// TIA Portal V20 export
FUNCTION "FC_Sequenza_Start" : Void   // FC300, LAD
{ S7_Optimized_Access := 'TRUE' }
// stored: AutoNumber false, SetENOAutomatically false
   VAR_TEMP   // added for the SCL form of the ladder/FBD networks
      _w1 : Bool;
      _w2 : Bool;
      _w3 : Bool;
      _w4 : Bool;
      _w5 : Bool;
      _w6 : Bool;
      _w7 : Bool;
      _w8 : Bool;
      _w9 : Bool;
      _w10 : Bool;
   END_VAR
BEGIN

REGION Network 1: Controllo ventilatori zona 1
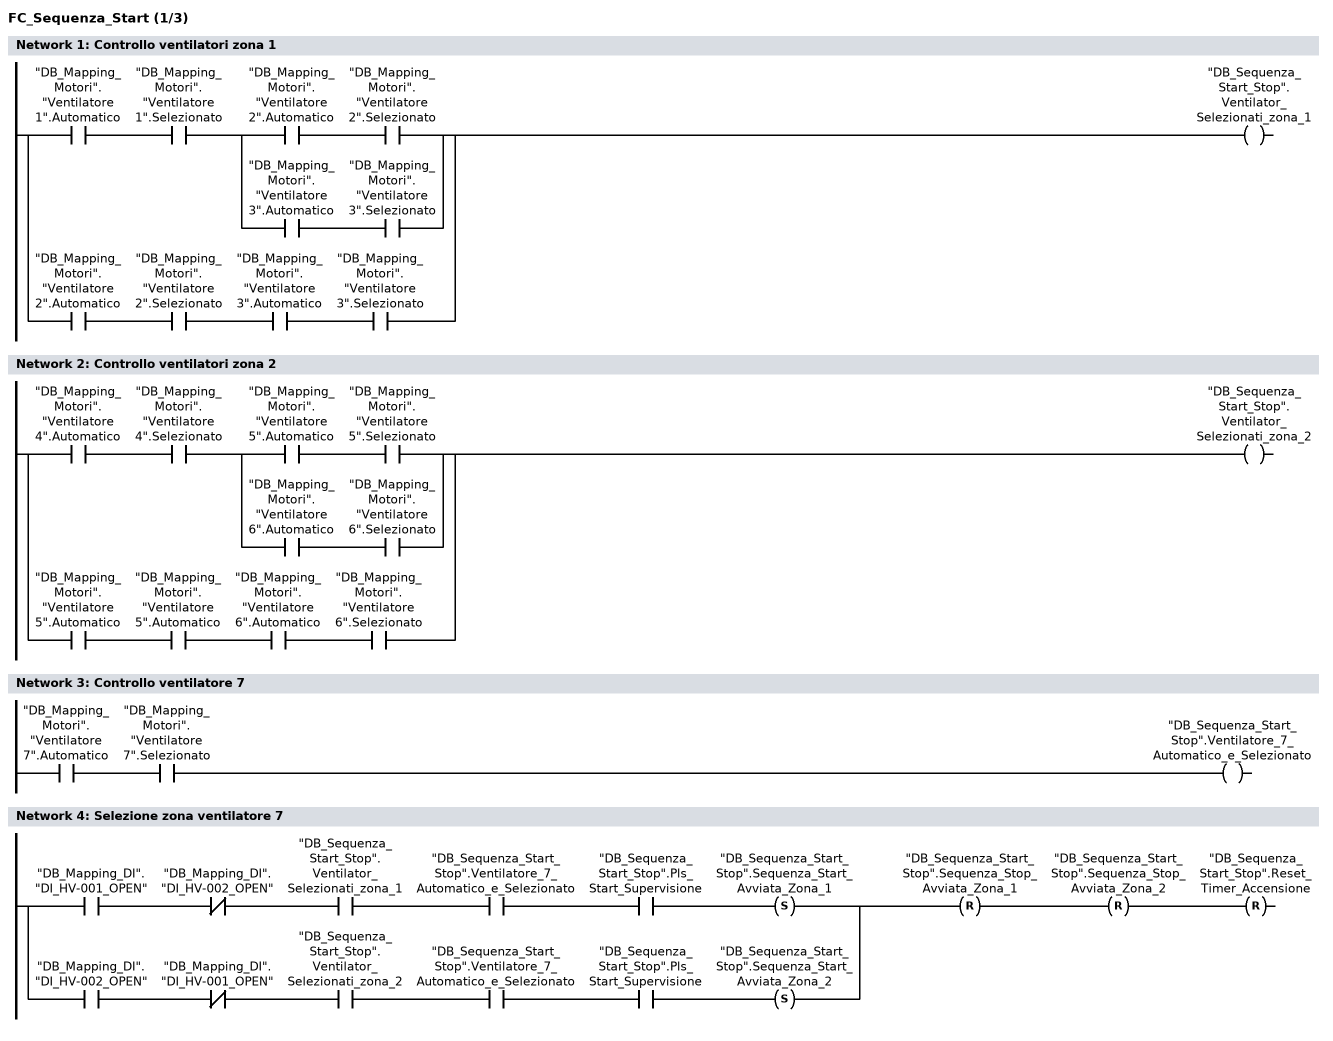
   RUNG wire#powerrail
      Contact( "DB_Mapping_Motori"."Ventilatore 1".Automatico )
      Contact( "DB_Mapping_Motori"."Ventilatore 1".Selezionato )
      wire#w1
      Contact( "DB_Mapping_Motori"."Ventilatore 2".Automatico )
      Contact( "DB_Mapping_Motori"."Ventilatore 2".Selezionato )
      wire#w2
      Coil( "DB_Sequenza_Start_Stop".Ventilator_Selezionati_zona_1 )
   END_RUNG
   RUNG wire#w1
      Contact( "DB_Mapping_Motori"."Ventilatore 3".Automatico )
      Contact( "DB_Mapping_Motori"."Ventilatore 3".Selezionato )
   END_RUNG wire#w2
   RUNG wire#powerrail
      Contact( "DB_Mapping_Motori"."Ventilatore 2".Automatico )
      Contact( "DB_Mapping_Motori"."Ventilatore 2".Selezionato )
      Contact( "DB_Mapping_Motori"."Ventilatore 3".Automatico )
      Contact( "DB_Mapping_Motori"."Ventilatore 3".Selezionato )
   END_RUNG wire#w2
   // the same network as SCL:
   "DB_Sequenza_Start_Stop".Ventilator_Selezionati_zona_1 := ("DB_Mapping_Motori"."Ventilatore 1".Automatico AND "DB_Mapping_Motori"."Ventilatore 1".Selezionato AND (("DB_Mapping_Motori"."Ventilatore 2".Automatico AND "DB_Mapping_Motori"."Ventilatore 2".Selezionato) OR ("DB_Mapping_Motori"."Ventilatore 3".Automatico AND "DB_Mapping_Motori"."Ventilatore 3".Selezionato))) OR ("DB_Mapping_Motori"."Ventilatore 2".Automatico AND "DB_Mapping_Motori"."Ventilatore 2".Selezionato AND "DB_Mapping_Motori"."Ventilatore 3".Automatico AND "DB_Mapping_Motori"."Ventilatore 3".Selezionato);
END_REGION

REGION Network 2: Controllo ventilatori zona 2
   RUNG wire#powerrail
      Contact( "DB_Mapping_Motori"."Ventilatore 4".Automatico )
      Contact( "DB_Mapping_Motori"."Ventilatore 4".Selezionato )
      wire#w1
      Contact( "DB_Mapping_Motori"."Ventilatore 5".Automatico )
      Contact( "DB_Mapping_Motori"."Ventilatore 5".Selezionato )
      wire#w2
      Coil( "DB_Sequenza_Start_Stop".Ventilator_Selezionati_zona_2 )
   END_RUNG
   RUNG wire#w1
      Contact( "DB_Mapping_Motori"."Ventilatore 6".Automatico )
      Contact( "DB_Mapping_Motori"."Ventilatore 6".Selezionato )
   END_RUNG wire#w2
   RUNG wire#powerrail
      Contact( "DB_Mapping_Motori"."Ventilatore 5".Automatico )
      Contact( "DB_Mapping_Motori"."Ventilatore 5".Automatico )
      Contact( "DB_Mapping_Motori"."Ventilatore 6".Automatico )
      Contact( "DB_Mapping_Motori"."Ventilatore 6".Selezionato )
   END_RUNG wire#w2
   // the same network as SCL:
   "DB_Sequenza_Start_Stop".Ventilator_Selezionati_zona_2 := ("DB_Mapping_Motori"."Ventilatore 4".Automatico AND "DB_Mapping_Motori"."Ventilatore 4".Selezionato AND (("DB_Mapping_Motori"."Ventilatore 5".Automatico AND "DB_Mapping_Motori"."Ventilatore 5".Selezionato) OR ("DB_Mapping_Motori"."Ventilatore 6".Automatico AND "DB_Mapping_Motori"."Ventilatore 6".Selezionato))) OR ("DB_Mapping_Motori"."Ventilatore 5".Automatico AND "DB_Mapping_Motori"."Ventilatore 5".Automatico AND "DB_Mapping_Motori"."Ventilatore 6".Automatico AND "DB_Mapping_Motori"."Ventilatore 6".Selezionato);
END_REGION

REGION Network 3: Controllo ventilatore 7
   RUNG wire#powerrail
      Contact( "DB_Mapping_Motori"."Ventilatore 7".Automatico )
      Contact( "DB_Mapping_Motori"."Ventilatore 7".Selezionato )
      Coil( "DB_Sequenza_Start_Stop".Ventilatore_7_Automatico_e_Selezionato )
   END_RUNG
   // the same network as SCL:
   "DB_Sequenza_Start_Stop".Ventilatore_7_Automatico_e_Selezionato := "DB_Mapping_Motori"."Ventilatore 7".Automatico AND "DB_Mapping_Motori"."Ventilatore 7".Selezionato;
END_REGION

REGION Network 4: Selezione zona ventilatore 7
   RUNG wire#powerrail
      Contact( "DB_Mapping_DI"."DI_HV-001_OPEN" )
      I_Contact( "DB_Mapping_DI"."DI_HV-002_OPEN" )
      Contact( "DB_Sequenza_Start_Stop".Ventilator_Selezionati_zona_1 )
      Contact( "DB_Sequenza_Start_Stop".Ventilatore_7_Automatico_e_Selezionato )
      Contact( "DB_Sequenza_Start_Stop".Pls_Start_Supervisione )
      S_Coil( "DB_Sequenza_Start_Stop".Sequenza_Start_Avviata_Zona_1 )
      wire#w1
      R_Coil( "DB_Sequenza_Start_Stop".Sequenza_Stop_Avviata_Zona_1 )
      R_Coil( "DB_Sequenza_Start_Stop".Sequenza_Stop_Avviata_Zona_2 )
      R_Coil( "DB_Sequenza_Start_Stop".Reset_Timer_Accensione )
   END_RUNG
   RUNG wire#powerrail
      Contact( "DB_Mapping_DI"."DI_HV-002_OPEN" )
      I_Contact( "DB_Mapping_DI"."DI_HV-001_OPEN" )
      Contact( "DB_Sequenza_Start_Stop".Ventilator_Selezionati_zona_2 )
      Contact( "DB_Sequenza_Start_Stop".Ventilatore_7_Automatico_e_Selezionato )
      Contact( "DB_Sequenza_Start_Stop".Pls_Start_Supervisione )
      S_Coil( "DB_Sequenza_Start_Stop".Sequenza_Start_Avviata_Zona_2 )
   END_RUNG wire#w1
   // the same network as SCL:
   #_w1 := "DB_Mapping_DI"."DI_HV-001_OPEN" AND NOT "DB_Mapping_DI"."DI_HV-002_OPEN" AND "DB_Sequenza_Start_Stop".Ventilator_Selezionati_zona_1 AND "DB_Sequenza_Start_Stop".Ventilatore_7_Automatico_e_Selezionato AND "DB_Sequenza_Start_Stop".Pls_Start_Supervisione;
   IF #_w1 THEN "DB_Sequenza_Start_Stop".Sequenza_Start_Avviata_Zona_1 := TRUE; END_IF;
   #_w2 := "DB_Mapping_DI"."DI_HV-002_OPEN" AND NOT "DB_Mapping_DI"."DI_HV-001_OPEN" AND "DB_Sequenza_Start_Stop".Ventilator_Selezionati_zona_2 AND "DB_Sequenza_Start_Stop".Ventilatore_7_Automatico_e_Selezionato AND "DB_Sequenza_Start_Stop".Pls_Start_Supervisione;
   IF #_w2 THEN "DB_Sequenza_Start_Stop".Sequenza_Start_Avviata_Zona_2 := TRUE; END_IF;
   IF #_w1 OR #_w2 THEN
       "DB_Sequenza_Start_Stop".Sequenza_Stop_Avviata_Zona_1 := FALSE;
       "DB_Sequenza_Start_Stop".Sequenza_Stop_Avviata_Zona_2 := FALSE;
       "DB_Sequenza_Start_Stop".Reset_Timer_Accensione := FALSE;
   END_IF;
END_REGION

REGION Network 5: Accensione ventilatori
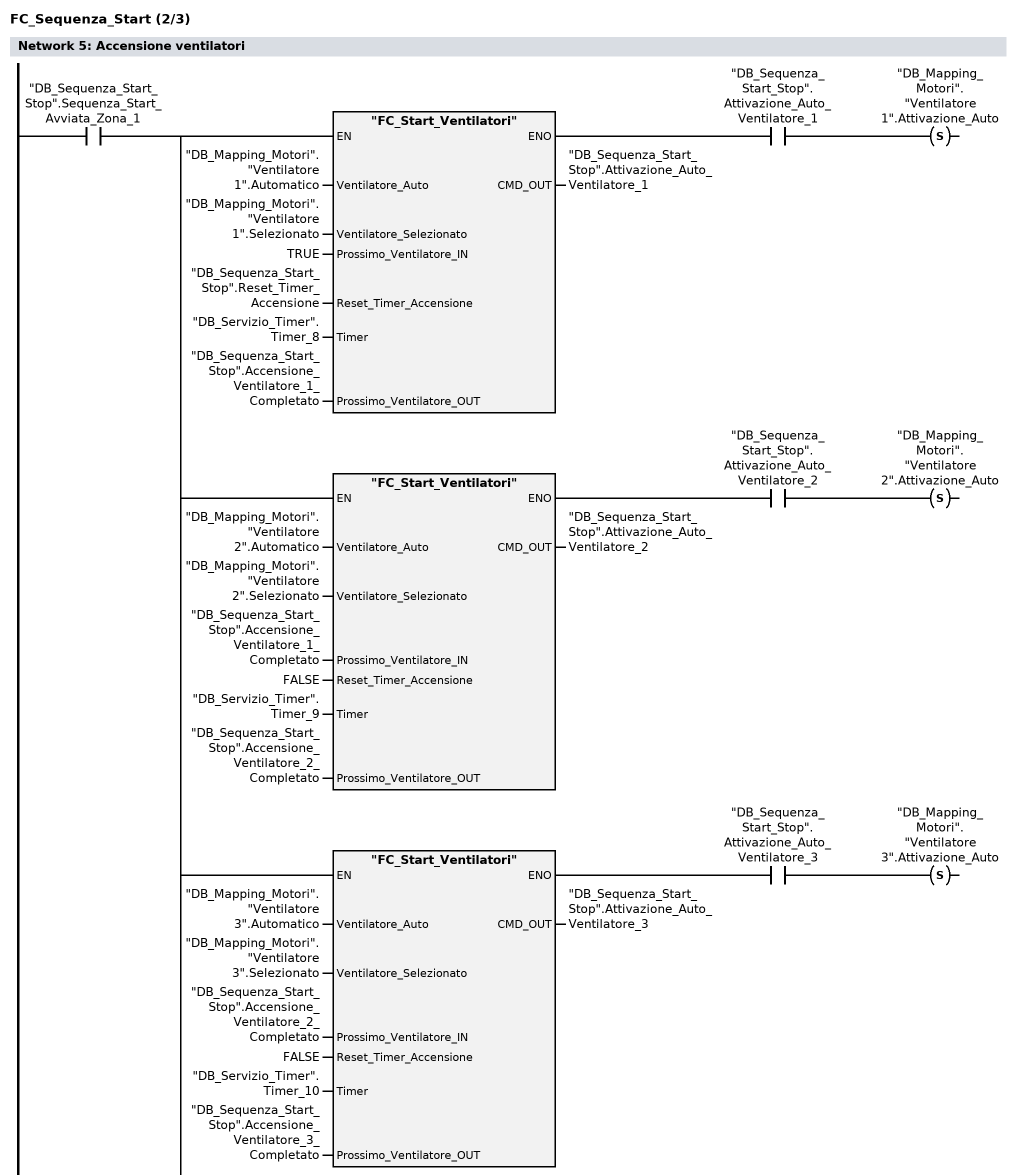
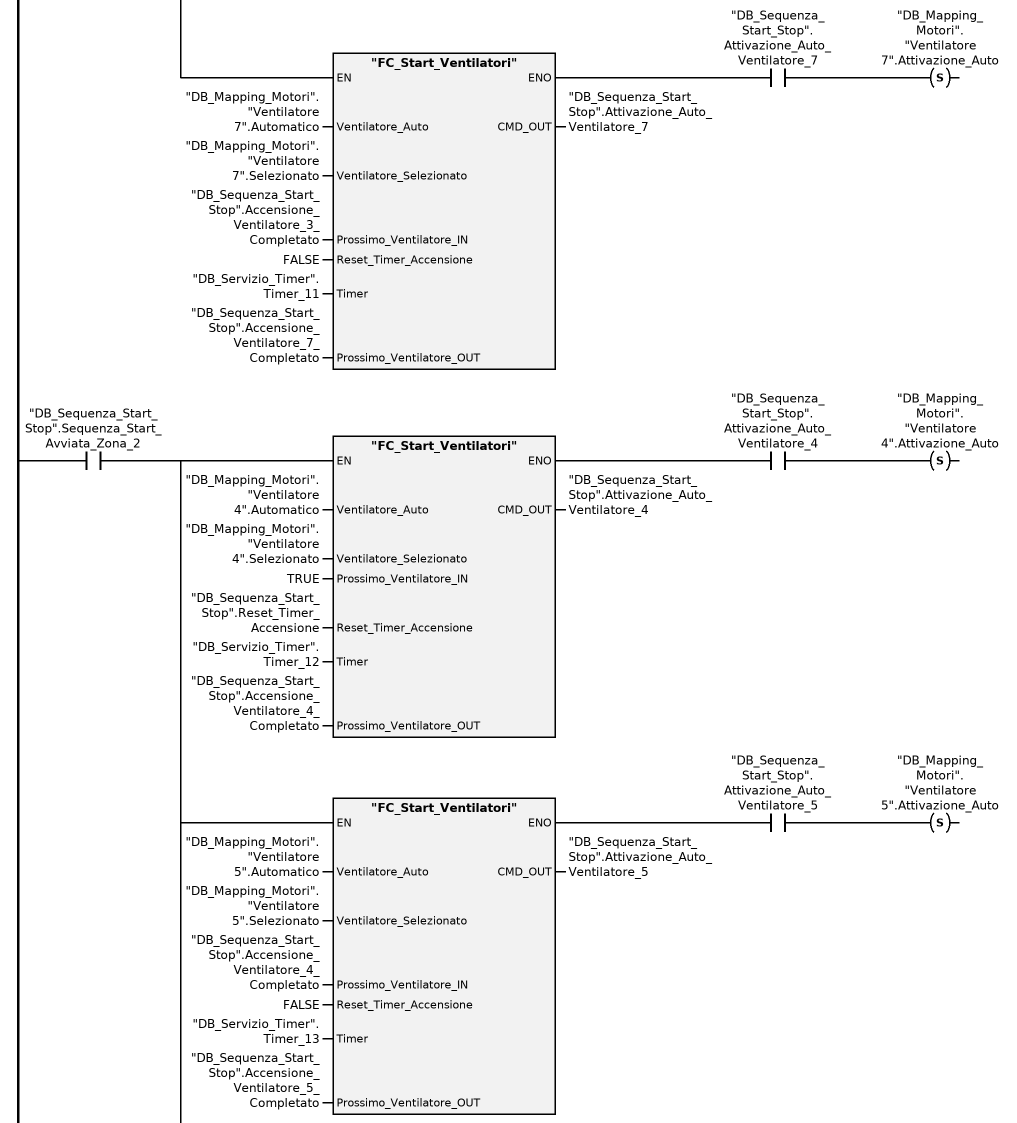
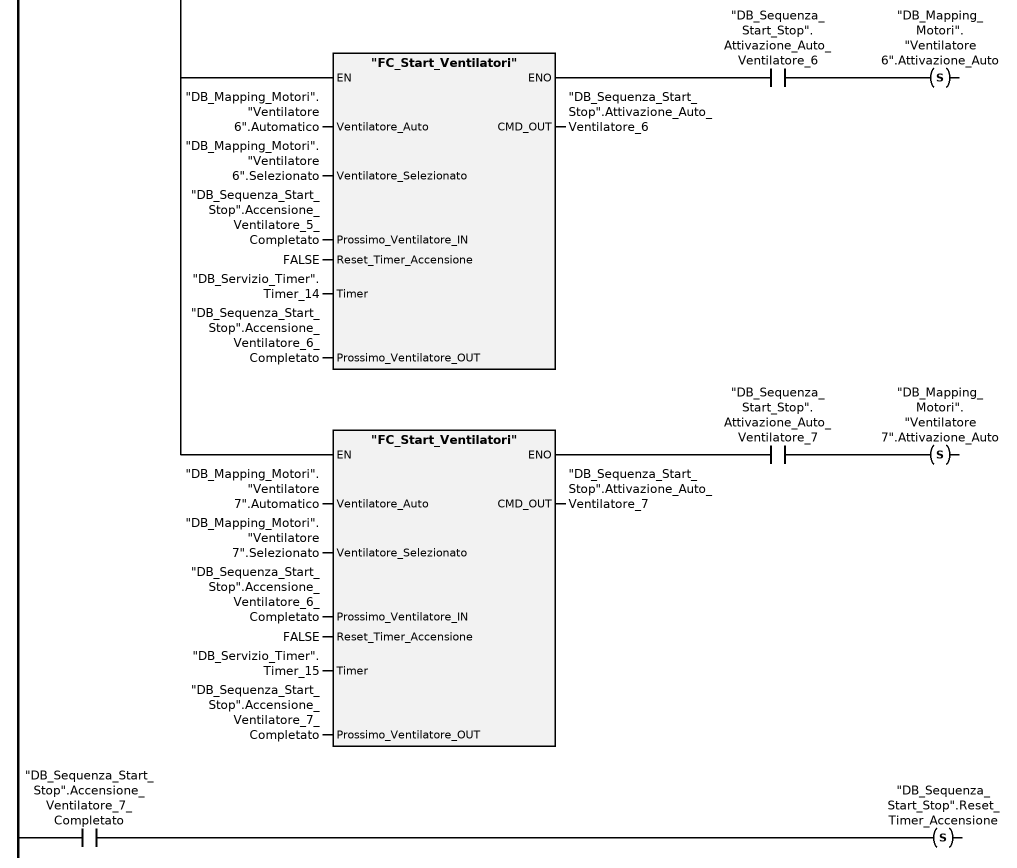
   RUNG wire#powerrail
      Contact( "DB_Sequenza_Start_Stop".Sequenza_Start_Avviata_Zona_1 )
      wire#w1
      "FC_Start_Ventilatori"(Ventilatore_Auto := "DB_Mapping_Motori"."Ventilatore 1".Automatico, Ventilatore_Selezionato := "DB_Mapping_Motori"."Ventilatore 1".Selezionato, Prossimo_Ventilatore_IN := TRUE, Reset_Timer_Accensione := "DB_Sequenza_Start_Stop".Reset_Timer_Accensione, "Timer" := "DB_Servizio_Timer".Timer_8, Prossimo_Ventilatore_OUT := "DB_Sequenza_Start_Stop".Accensione_Ventilatore_1_Completato, CMD_OUT => "DB_Sequenza_Start_Stop".Attivazione_Auto_Ventilatore_1)
      Contact( "DB_Sequenza_Start_Stop".Attivazione_Auto_Ventilatore_1 )
      S_Coil( "DB_Mapping_Motori"."Ventilatore 1".Attivazione_Auto )
   END_RUNG
   RUNG wire#w1
      "FC_Start_Ventilatori"(Ventilatore_Auto := "DB_Mapping_Motori"."Ventilatore 2".Automatico, Ventilatore_Selezionato := "DB_Mapping_Motori"."Ventilatore 2".Selezionato, Prossimo_Ventilatore_IN := "DB_Sequenza_Start_Stop".Accensione_Ventilatore_1_Completato, Reset_Timer_Accensione := FALSE, "Timer" := "DB_Servizio_Timer".Timer_9, Prossimo_Ventilatore_OUT := "DB_Sequenza_Start_Stop".Accensione_Ventilatore_2_Completato, CMD_OUT => "DB_Sequenza_Start_Stop".Attivazione_Auto_Ventilatore_2)
      Contact( "DB_Sequenza_Start_Stop".Attivazione_Auto_Ventilatore_2 )
      S_Coil( "DB_Mapping_Motori"."Ventilatore 2".Attivazione_Auto )
   END_RUNG
   RUNG wire#w1
      "FC_Start_Ventilatori"(Ventilatore_Auto := "DB_Mapping_Motori"."Ventilatore 3".Automatico, Ventilatore_Selezionato := "DB_Mapping_Motori"."Ventilatore 3".Selezionato, Prossimo_Ventilatore_IN := "DB_Sequenza_Start_Stop".Accensione_Ventilatore_2_Completato, Reset_Timer_Accensione := FALSE, "Timer" := "DB_Servizio_Timer".Timer_10, Prossimo_Ventilatore_OUT := "DB_Sequenza_Start_Stop".Accensione_Ventilatore_3_Completato, CMD_OUT => "DB_Sequenza_Start_Stop".Attivazione_Auto_Ventilatore_3)
      Contact( "DB_Sequenza_Start_Stop".Attivazione_Auto_Ventilatore_3 )
      S_Coil( "DB_Mapping_Motori"."Ventilatore 3".Attivazione_Auto )
   END_RUNG
   RUNG wire#w1
      "FC_Start_Ventilatori"(Ventilatore_Auto := "DB_Mapping_Motori"."Ventilatore 7".Automatico, Ventilatore_Selezionato := "DB_Mapping_Motori"."Ventilatore 7".Selezionato, Prossimo_Ventilatore_IN := "DB_Sequenza_Start_Stop".Accensione_Ventilatore_3_Completato, Reset_Timer_Accensione := FALSE, "Timer" := "DB_Servizio_Timer".Timer_11, Prossimo_Ventilatore_OUT := "DB_Sequenza_Start_Stop".Accensione_Ventilatore_7_Completato, CMD_OUT => "DB_Sequenza_Start_Stop".Attivazione_Auto_Ventilatore_7)
      Contact( "DB_Sequenza_Start_Stop".Attivazione_Auto_Ventilatore_7 )
      S_Coil( "DB_Mapping_Motori"."Ventilatore 7".Attivazione_Auto )
   END_RUNG
   RUNG wire#powerrail
      Contact( "DB_Sequenza_Start_Stop".Sequenza_Start_Avviata_Zona_2 )
      wire#w2
      "FC_Start_Ventilatori"(Ventilatore_Auto := "DB_Mapping_Motori"."Ventilatore 4".Automatico, Ventilatore_Selezionato := "DB_Mapping_Motori"."Ventilatore 4".Selezionato, Prossimo_Ventilatore_IN := TRUE, Reset_Timer_Accensione := "DB_Sequenza_Start_Stop".Reset_Timer_Accensione, "Timer" := "DB_Servizio_Timer".Timer_12, Prossimo_Ventilatore_OUT := "DB_Sequenza_Start_Stop".Accensione_Ventilatore_4_Completato, CMD_OUT => "DB_Sequenza_Start_Stop".Attivazione_Auto_Ventilatore_4)
      Contact( "DB_Sequenza_Start_Stop".Attivazione_Auto_Ventilatore_4 )
      S_Coil( "DB_Mapping_Motori"."Ventilatore 4".Attivazione_Auto )
   END_RUNG
   RUNG wire#w2
      "FC_Start_Ventilatori"(Ventilatore_Auto := "DB_Mapping_Motori"."Ventilatore 5".Automatico, Ventilatore_Selezionato := "DB_Mapping_Motori"."Ventilatore 5".Selezionato, Prossimo_Ventilatore_IN := "DB_Sequenza_Start_Stop".Accensione_Ventilatore_4_Completato, Reset_Timer_Accensione := FALSE, "Timer" := "DB_Servizio_Timer".Timer_13, Prossimo_Ventilatore_OUT := "DB_Sequenza_Start_Stop".Accensione_Ventilatore_5_Completato, CMD_OUT => "DB_Sequenza_Start_Stop".Attivazione_Auto_Ventilatore_5)
      Contact( "DB_Sequenza_Start_Stop".Attivazione_Auto_Ventilatore_5 )
      S_Coil( "DB_Mapping_Motori"."Ventilatore 5".Attivazione_Auto )
   END_RUNG
   RUNG wire#w2
      "FC_Start_Ventilatori"(Ventilatore_Auto := "DB_Mapping_Motori"."Ventilatore 6".Automatico, Ventilatore_Selezionato := "DB_Mapping_Motori"."Ventilatore 6".Selezionato, Prossimo_Ventilatore_IN := "DB_Sequenza_Start_Stop".Accensione_Ventilatore_5_Completato, Reset_Timer_Accensione := FALSE, "Timer" := "DB_Servizio_Timer".Timer_14, Prossimo_Ventilatore_OUT := "DB_Sequenza_Start_Stop".Accensione_Ventilatore_6_Completato, CMD_OUT => "DB_Sequenza_Start_Stop".Attivazione_Auto_Ventilatore_6)
      Contact( "DB_Sequenza_Start_Stop".Attivazione_Auto_Ventilatore_6 )
      S_Coil( "DB_Mapping_Motori"."Ventilatore 6".Attivazione_Auto )
   END_RUNG
   RUNG wire#w2
      "FC_Start_Ventilatori"(Ventilatore_Auto := "DB_Mapping_Motori"."Ventilatore 7".Automatico, Ventilatore_Selezionato := "DB_Mapping_Motori"."Ventilatore 7".Selezionato, Prossimo_Ventilatore_IN := "DB_Sequenza_Start_Stop".Accensione_Ventilatore_6_Completato, Reset_Timer_Accensione := FALSE, "Timer" := "DB_Servizio_Timer".Timer_15, Prossimo_Ventilatore_OUT := "DB_Sequenza_Start_Stop".Accensione_Ventilatore_7_Completato, CMD_OUT => "DB_Sequenza_Start_Stop".Attivazione_Auto_Ventilatore_7)
      Contact( "DB_Sequenza_Start_Stop".Attivazione_Auto_Ventilatore_7 )
      S_Coil( "DB_Mapping_Motori"."Ventilatore 7".Attivazione_Auto )
   END_RUNG
   RUNG wire#powerrail
      Contact( "DB_Sequenza_Start_Stop".Accensione_Ventilatore_7_Completato )
      S_Coil( "DB_Sequenza_Start_Stop".Reset_Timer_Accensione )
   END_RUNG
   // the same network as SCL:
   #_w2 := "DB_Sequenza_Start_Stop".Sequenza_Start_Avviata_Zona_1;
   "FC_Start_Ventilatori"(EN := "DB_Sequenza_Start_Stop".Sequenza_Start_Avviata_Zona_1,
                          Ventilatore_Auto := "DB_Mapping_Motori"."Ventilatore 1".Automatico,
                          Ventilatore_Selezionato := "DB_Mapping_Motori"."Ventilatore 1".Selezionato,
                          Prossimo_Ventilatore_IN := TRUE,
                          Reset_Timer_Accensione := "DB_Sequenza_Start_Stop".Reset_Timer_Accensione,
                          "Timer" := "DB_Servizio_Timer".Timer_8,
                          Prossimo_Ventilatore_OUT := "DB_Sequenza_Start_Stop".Accensione_Ventilatore_1_Completato,
                          CMD_OUT => "DB_Sequenza_Start_Stop".Attivazione_Auto_Ventilatore_1,
                          ENO => #_w1);
   IF #_w1 AND "DB_Sequenza_Start_Stop".Attivazione_Auto_Ventilatore_1 THEN
       "DB_Mapping_Motori"."Ventilatore 1".Attivazione_Auto := TRUE;
   END_IF;
   "FC_Start_Ventilatori"(EN := #_w2,
                          Ventilatore_Auto := "DB_Mapping_Motori"."Ventilatore 2".Automatico,
                          Ventilatore_Selezionato := "DB_Mapping_Motori"."Ventilatore 2".Selezionato,
                          Prossimo_Ventilatore_IN := "DB_Sequenza_Start_Stop".Accensione_Ventilatore_1_Completato,
                          Reset_Timer_Accensione := FALSE,
                          "Timer" := "DB_Servizio_Timer".Timer_9,
                          Prossimo_Ventilatore_OUT := "DB_Sequenza_Start_Stop".Accensione_Ventilatore_2_Completato,
                          CMD_OUT => "DB_Sequenza_Start_Stop".Attivazione_Auto_Ventilatore_2,
                          ENO => #_w3);
   IF #_w3 AND "DB_Sequenza_Start_Stop".Attivazione_Auto_Ventilatore_2 THEN
       "DB_Mapping_Motori"."Ventilatore 2".Attivazione_Auto := TRUE;
   END_IF;
   "FC_Start_Ventilatori"(EN := #_w2,
                          Ventilatore_Auto := "DB_Mapping_Motori"."Ventilatore 3".Automatico,
                          Ventilatore_Selezionato := "DB_Mapping_Motori"."Ventilatore 3".Selezionato,
                          Prossimo_Ventilatore_IN := "DB_Sequenza_Start_Stop".Accensione_Ventilatore_2_Completato,
                          Reset_Timer_Accensione := FALSE,
                          "Timer" := "DB_Servizio_Timer".Timer_10,
                          Prossimo_Ventilatore_OUT := "DB_Sequenza_Start_Stop".Accensione_Ventilatore_3_Completato,
                          CMD_OUT => "DB_Sequenza_Start_Stop".Attivazione_Auto_Ventilatore_3,
                          ENO => #_w4);
   IF #_w4 AND "DB_Sequenza_Start_Stop".Attivazione_Auto_Ventilatore_3 THEN
       "DB_Mapping_Motori"."Ventilatore 3".Attivazione_Auto := TRUE;
   END_IF;
   "FC_Start_Ventilatori"(EN := #_w2,
                          Ventilatore_Auto := "DB_Mapping_Motori"."Ventilatore 7".Automatico,
                          Ventilatore_Selezionato := "DB_Mapping_Motori"."Ventilatore 7".Selezionato,
                          Prossimo_Ventilatore_IN := "DB_Sequenza_Start_Stop".Accensione_Ventilatore_3_Completato,
                          Reset_Timer_Accensione := FALSE,
                          "Timer" := "DB_Servizio_Timer".Timer_11,
                          Prossimo_Ventilatore_OUT := "DB_Sequenza_Start_Stop".Accensione_Ventilatore_7_Completato,
                          CMD_OUT => "DB_Sequenza_Start_Stop".Attivazione_Auto_Ventilatore_7,
                          ENO => #_w5);
   IF #_w5 AND "DB_Sequenza_Start_Stop".Attivazione_Auto_Ventilatore_7 THEN
       "DB_Mapping_Motori"."Ventilatore 7".Attivazione_Auto := TRUE;
   END_IF;
   #_w7 := "DB_Sequenza_Start_Stop".Sequenza_Start_Avviata_Zona_2;
   "FC_Start_Ventilatori"(EN := "DB_Sequenza_Start_Stop".Sequenza_Start_Avviata_Zona_2,
                          Ventilatore_Auto := "DB_Mapping_Motori"."Ventilatore 4".Automatico,
                          Ventilatore_Selezionato := "DB_Mapping_Motori"."Ventilatore 4".Selezionato,
                          Prossimo_Ventilatore_IN := TRUE,
                          Reset_Timer_Accensione := "DB_Sequenza_Start_Stop".Reset_Timer_Accensione,
                          "Timer" := "DB_Servizio_Timer".Timer_12,
                          Prossimo_Ventilatore_OUT := "DB_Sequenza_Start_Stop".Accensione_Ventilatore_4_Completato,
                          CMD_OUT => "DB_Sequenza_Start_Stop".Attivazione_Auto_Ventilatore_4,
                          ENO => #_w6);
   IF #_w6 AND "DB_Sequenza_Start_Stop".Attivazione_Auto_Ventilatore_4 THEN
       "DB_Mapping_Motori"."Ventilatore 4".Attivazione_Auto := TRUE;
   END_IF;
   "FC_Start_Ventilatori"(EN := #_w7,
                          Ventilatore_Auto := "DB_Mapping_Motori"."Ventilatore 5".Automatico,
                          Ventilatore_Selezionato := "DB_Mapping_Motori"."Ventilatore 5".Selezionato,
                          Prossimo_Ventilatore_IN := "DB_Sequenza_Start_Stop".Accensione_Ventilatore_4_Completato,
                          Reset_Timer_Accensione := FALSE,
                          "Timer" := "DB_Servizio_Timer".Timer_13,
                          Prossimo_Ventilatore_OUT := "DB_Sequenza_Start_Stop".Accensione_Ventilatore_5_Completato,
                          CMD_OUT => "DB_Sequenza_Start_Stop".Attivazione_Auto_Ventilatore_5,
                          ENO => #_w8);
   IF #_w8 AND "DB_Sequenza_Start_Stop".Attivazione_Auto_Ventilatore_5 THEN
       "DB_Mapping_Motori"."Ventilatore 5".Attivazione_Auto := TRUE;
   END_IF;
   "FC_Start_Ventilatori"(EN := #_w7,
                          Ventilatore_Auto := "DB_Mapping_Motori"."Ventilatore 6".Automatico,
                          Ventilatore_Selezionato := "DB_Mapping_Motori"."Ventilatore 6".Selezionato,
                          Prossimo_Ventilatore_IN := "DB_Sequenza_Start_Stop".Accensione_Ventilatore_5_Completato,
                          Reset_Timer_Accensione := FALSE,
                          "Timer" := "DB_Servizio_Timer".Timer_14,
                          Prossimo_Ventilatore_OUT := "DB_Sequenza_Start_Stop".Accensione_Ventilatore_6_Completato,
                          CMD_OUT => "DB_Sequenza_Start_Stop".Attivazione_Auto_Ventilatore_6,
                          ENO => #_w9);
   IF #_w9 AND "DB_Sequenza_Start_Stop".Attivazione_Auto_Ventilatore_6 THEN
       "DB_Mapping_Motori"."Ventilatore 6".Attivazione_Auto := TRUE;
   END_IF;
   "FC_Start_Ventilatori"(EN := #_w7,
                          Ventilatore_Auto := "DB_Mapping_Motori"."Ventilatore 7".Automatico,
                          Ventilatore_Selezionato := "DB_Mapping_Motori"."Ventilatore 7".Selezionato,
                          Prossimo_Ventilatore_IN := "DB_Sequenza_Start_Stop".Accensione_Ventilatore_6_Completato,
                          Reset_Timer_Accensione := FALSE,
                          "Timer" := "DB_Servizio_Timer".Timer_15,
                          Prossimo_Ventilatore_OUT := "DB_Sequenza_Start_Stop".Accensione_Ventilatore_7_Completato,
                          CMD_OUT => "DB_Sequenza_Start_Stop".Attivazione_Auto_Ventilatore_7,
                          ENO => #_w10);
   IF #_w10 AND "DB_Sequenza_Start_Stop".Attivazione_Auto_Ventilatore_7 THEN
       "DB_Mapping_Motori"."Ventilatore 7".Attivazione_Auto := TRUE;
   END_IF;
   IF "DB_Sequenza_Start_Stop".Accensione_Ventilatore_7_Completato THEN
       "DB_Sequenza_Start_Stop".Reset_Timer_Accensione := TRUE;
   END_IF;
END_REGION

REGION Network 6: Gestione avvio pompe a sequenza attiva
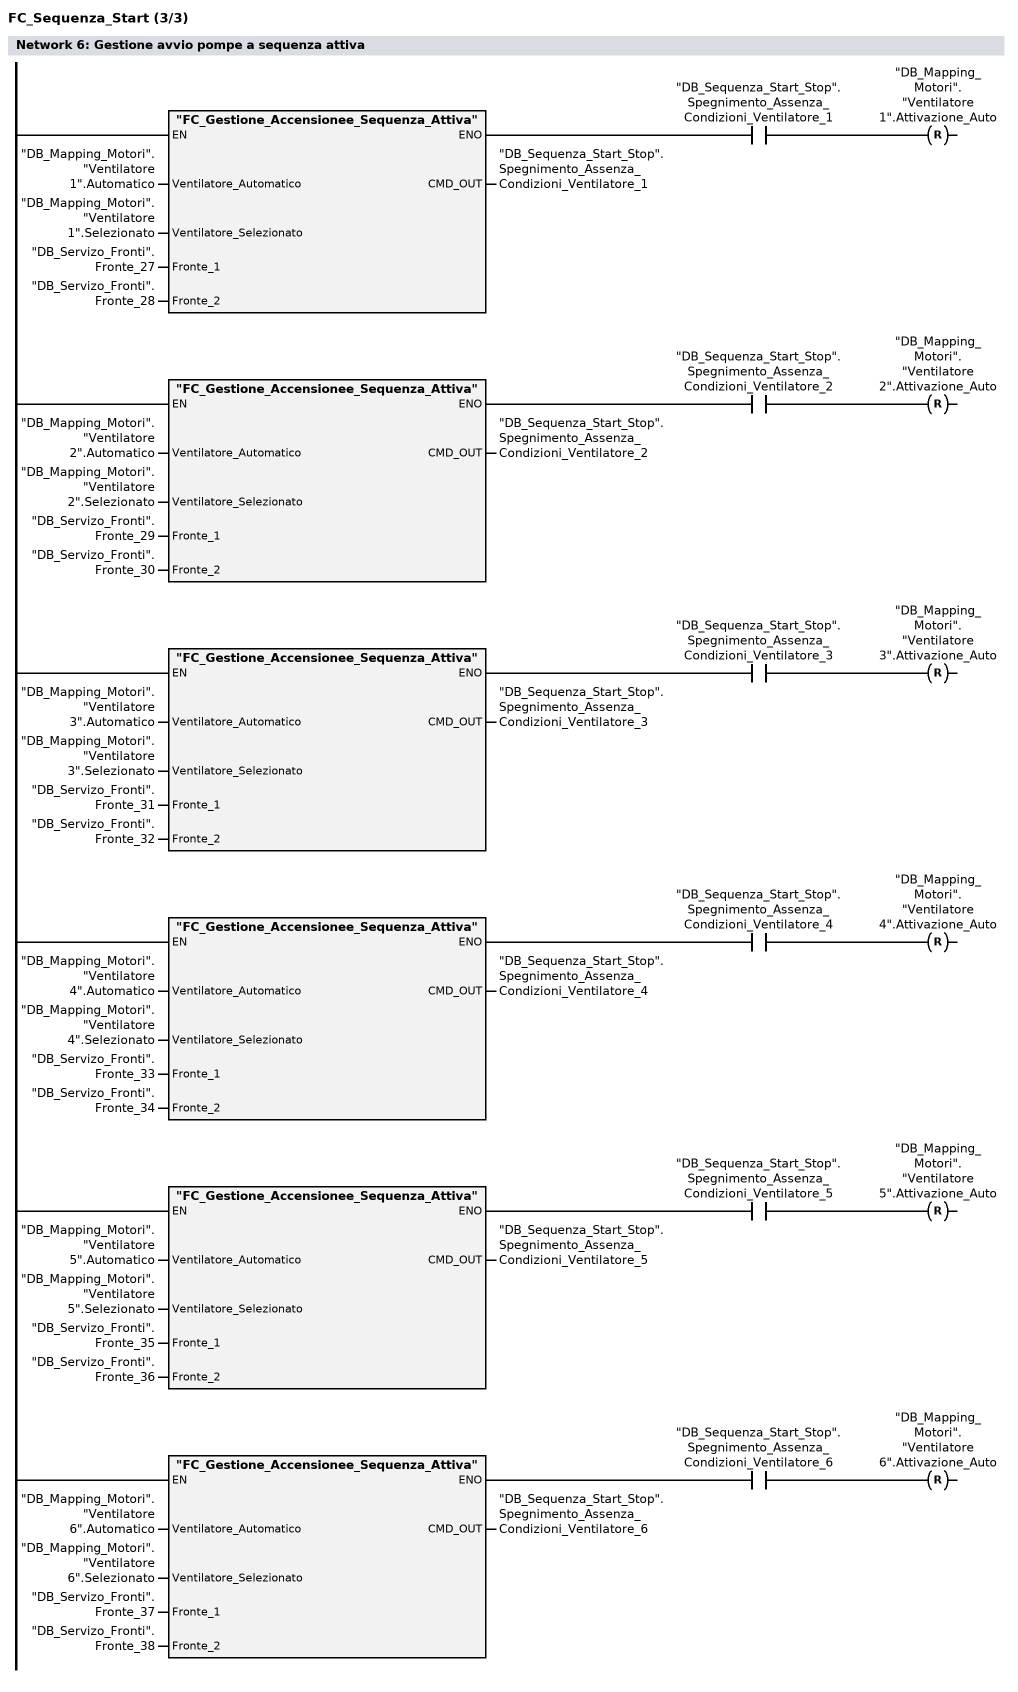
   RUNG wire#powerrail
      "FC_Gestione_Accensionee_Sequenza_Attiva"(Ventilatore_Automatico := "DB_Mapping_Motori"."Ventilatore 1".Automatico, Ventilatore_Selezionato := "DB_Mapping_Motori"."Ventilatore 1".Selezionato, Fronte_1 := "DB_Servizo_Fronti".Fronte_27, Fronte_2 := "DB_Servizo_Fronti".Fronte_28, CMD_OUT => "DB_Sequenza_Start_Stop".Spegnimento_Assenza_Condizioni_Ventilatore_1)
      Contact( "DB_Sequenza_Start_Stop".Spegnimento_Assenza_Condizioni_Ventilatore_1 )
      R_Coil( "DB_Mapping_Motori"."Ventilatore 1".Attivazione_Auto )
   END_RUNG
   RUNG wire#powerrail
      "FC_Gestione_Accensionee_Sequenza_Attiva"(Ventilatore_Automatico := "DB_Mapping_Motori"."Ventilatore 2".Automatico, Ventilatore_Selezionato := "DB_Mapping_Motori"."Ventilatore 2".Selezionato, Fronte_1 := "DB_Servizo_Fronti".Fronte_29, Fronte_2 := "DB_Servizo_Fronti".Fronte_30, CMD_OUT => "DB_Sequenza_Start_Stop".Spegnimento_Assenza_Condizioni_Ventilatore_2)
      Contact( "DB_Sequenza_Start_Stop".Spegnimento_Assenza_Condizioni_Ventilatore_2 )
      R_Coil( "DB_Mapping_Motori"."Ventilatore 2".Attivazione_Auto )
   END_RUNG
   RUNG wire#powerrail
      "FC_Gestione_Accensionee_Sequenza_Attiva"(Ventilatore_Automatico := "DB_Mapping_Motori"."Ventilatore 3".Automatico, Ventilatore_Selezionato := "DB_Mapping_Motori"."Ventilatore 3".Selezionato, Fronte_1 := "DB_Servizo_Fronti".Fronte_31, Fronte_2 := "DB_Servizo_Fronti".Fronte_32, CMD_OUT => "DB_Sequenza_Start_Stop".Spegnimento_Assenza_Condizioni_Ventilatore_3)
      Contact( "DB_Sequenza_Start_Stop".Spegnimento_Assenza_Condizioni_Ventilatore_3 )
      R_Coil( "DB_Mapping_Motori"."Ventilatore 3".Attivazione_Auto )
   END_RUNG
   RUNG wire#powerrail
      "FC_Gestione_Accensionee_Sequenza_Attiva"(Ventilatore_Automatico := "DB_Mapping_Motori"."Ventilatore 4".Automatico, Ventilatore_Selezionato := "DB_Mapping_Motori"."Ventilatore 4".Selezionato, Fronte_1 := "DB_Servizo_Fronti".Fronte_33, Fronte_2 := "DB_Servizo_Fronti".Fronte_34, CMD_OUT => "DB_Sequenza_Start_Stop".Spegnimento_Assenza_Condizioni_Ventilatore_4)
      Contact( "DB_Sequenza_Start_Stop".Spegnimento_Assenza_Condizioni_Ventilatore_4 )
      R_Coil( "DB_Mapping_Motori"."Ventilatore 4".Attivazione_Auto )
   END_RUNG
   RUNG wire#powerrail
      "FC_Gestione_Accensionee_Sequenza_Attiva"(Ventilatore_Automatico := "DB_Mapping_Motori"."Ventilatore 5".Automatico, Ventilatore_Selezionato := "DB_Mapping_Motori"."Ventilatore 5".Selezionato, Fronte_1 := "DB_Servizo_Fronti".Fronte_35, Fronte_2 := "DB_Servizo_Fronti".Fronte_36, CMD_OUT => "DB_Sequenza_Start_Stop".Spegnimento_Assenza_Condizioni_Ventilatore_5)
      Contact( "DB_Sequenza_Start_Stop".Spegnimento_Assenza_Condizioni_Ventilatore_5 )
      R_Coil( "DB_Mapping_Motori"."Ventilatore 5".Attivazione_Auto )
   END_RUNG
   RUNG wire#powerrail
      "FC_Gestione_Accensionee_Sequenza_Attiva"(Ventilatore_Automatico := "DB_Mapping_Motori"."Ventilatore 6".Automatico, Ventilatore_Selezionato := "DB_Mapping_Motori"."Ventilatore 6".Selezionato, Fronte_1 := "DB_Servizo_Fronti".Fronte_37, Fronte_2 := "DB_Servizo_Fronti".Fronte_38, CMD_OUT => "DB_Sequenza_Start_Stop".Spegnimento_Assenza_Condizioni_Ventilatore_6)
      Contact( "DB_Sequenza_Start_Stop".Spegnimento_Assenza_Condizioni_Ventilatore_6 )
      R_Coil( "DB_Mapping_Motori"."Ventilatore 6".Attivazione_Auto )
   END_RUNG
   // the same network as SCL:
   "FC_Gestione_Accensionee_Sequenza_Attiva"(Ventilatore_Automatico := "DB_Mapping_Motori"."Ventilatore 1".Automatico,
                           Ventilatore_Selezionato := "DB_Mapping_Motori"."Ventilatore 1".Selezionato,
                           Fronte_1 := "DB_Servizo_Fronti".Fronte_27,
                           Fronte_2 := "DB_Servizo_Fronti".Fronte_28,
                           CMD_OUT => "DB_Sequenza_Start_Stop".Spegnimento_Assenza_Condizioni_Ventilatore_1,
                           ENO => #_w1);
   IF #_w1 AND "DB_Sequenza_Start_Stop".Spegnimento_Assenza_Condizioni_Ventilatore_1 THEN
       "DB_Mapping_Motori"."Ventilatore 1".Attivazione_Auto := FALSE;
   END_IF;
   "FC_Gestione_Accensionee_Sequenza_Attiva"(Ventilatore_Automatico := "DB_Mapping_Motori"."Ventilatore 2".Automatico,
                           Ventilatore_Selezionato := "DB_Mapping_Motori"."Ventilatore 2".Selezionato,
                           Fronte_1 := "DB_Servizo_Fronti".Fronte_29,
                           Fronte_2 := "DB_Servizo_Fronti".Fronte_30,
                           CMD_OUT => "DB_Sequenza_Start_Stop".Spegnimento_Assenza_Condizioni_Ventilatore_2,
                           ENO => #_w2);
   IF #_w2 AND "DB_Sequenza_Start_Stop".Spegnimento_Assenza_Condizioni_Ventilatore_2 THEN
       "DB_Mapping_Motori"."Ventilatore 2".Attivazione_Auto := FALSE;
   END_IF;
   "FC_Gestione_Accensionee_Sequenza_Attiva"(Ventilatore_Automatico := "DB_Mapping_Motori"."Ventilatore 3".Automatico,
                           Ventilatore_Selezionato := "DB_Mapping_Motori"."Ventilatore 3".Selezionato,
                           Fronte_1 := "DB_Servizo_Fronti".Fronte_31,
                           Fronte_2 := "DB_Servizo_Fronti".Fronte_32,
                           CMD_OUT => "DB_Sequenza_Start_Stop".Spegnimento_Assenza_Condizioni_Ventilatore_3,
                           ENO => #_w3);
   IF #_w3 AND "DB_Sequenza_Start_Stop".Spegnimento_Assenza_Condizioni_Ventilatore_3 THEN
       "DB_Mapping_Motori"."Ventilatore 3".Attivazione_Auto := FALSE;
   END_IF;
   "FC_Gestione_Accensionee_Sequenza_Attiva"(Ventilatore_Automatico := "DB_Mapping_Motori"."Ventilatore 4".Automatico,
                           Ventilatore_Selezionato := "DB_Mapping_Motori"."Ventilatore 4".Selezionato,
                           Fronte_1 := "DB_Servizo_Fronti".Fronte_33,
                           Fronte_2 := "DB_Servizo_Fronti".Fronte_34,
                           CMD_OUT => "DB_Sequenza_Start_Stop".Spegnimento_Assenza_Condizioni_Ventilatore_4,
                           ENO => #_w4);
   IF #_w4 AND "DB_Sequenza_Start_Stop".Spegnimento_Assenza_Condizioni_Ventilatore_4 THEN
       "DB_Mapping_Motori"."Ventilatore 4".Attivazione_Auto := FALSE;
   END_IF;
   "FC_Gestione_Accensionee_Sequenza_Attiva"(Ventilatore_Automatico := "DB_Mapping_Motori"."Ventilatore 5".Automatico,
                           Ventilatore_Selezionato := "DB_Mapping_Motori"."Ventilatore 5".Selezionato,
                           Fronte_1 := "DB_Servizo_Fronti".Fronte_35,
                           Fronte_2 := "DB_Servizo_Fronti".Fronte_36,
                           CMD_OUT => "DB_Sequenza_Start_Stop".Spegnimento_Assenza_Condizioni_Ventilatore_5,
                           ENO => #_w5);
   IF #_w5 AND "DB_Sequenza_Start_Stop".Spegnimento_Assenza_Condizioni_Ventilatore_5 THEN
       "DB_Mapping_Motori"."Ventilatore 5".Attivazione_Auto := FALSE;
   END_IF;
   "FC_Gestione_Accensionee_Sequenza_Attiva"(Ventilatore_Automatico := "DB_Mapping_Motori"."Ventilatore 6".Automatico,
                           Ventilatore_Selezionato := "DB_Mapping_Motori"."Ventilatore 6".Selezionato,
                           Fronte_1 := "DB_Servizo_Fronti".Fronte_37,
                           Fronte_2 := "DB_Servizo_Fronti".Fronte_38,
                           CMD_OUT => "DB_Sequenza_Start_Stop".Spegnimento_Assenza_Condizioni_Ventilatore_6,
                           ENO => #_w6);
   IF #_w6 AND "DB_Sequenza_Start_Stop".Spegnimento_Assenza_Condizioni_Ventilatore_6 THEN
       "DB_Mapping_Motori"."Ventilatore 6".Attivazione_Auto := FALSE;
   END_IF;
END_REGION
END_FUNCTION
